// TIA Portal V20 export
TYPE "typeSequenceControlNodeHomeCheck_sideTapeFixStage"
// stored: Namespace Unit1.Em4
   STRUCT
      tape1PosPartNoDetect { ExternalWritable := 'False'} : Bool;
      tape1PosPartDetect { ExternalWritable := 'False'} : Bool;
      tape2PosPartDetect { ExternalWritable := 'False'} : Bool;
      tape3PosPartDetect { ExternalWritable := 'False'} : Bool;
      tape4PosPartDetect { ExternalWritable := 'False'} : Bool;
   END_STRUCT;
END_TYPE
